// Device/Application/CheckFunctions/CheckBounds
// Short description:      Test function to increase machine safety by checking for unauthorized array indices accesses.
// 
// Functional description: This function is implicitly called prior to each array access and verifies if the access is within the valid array bounds.
//                         If the access is authorized, the function returns the index to the calling POU and the access is completed.
//                         If the access is unauthorized, an exception is triggered as default error reaction. This exception results in an application stop and the system is set to safe state. 
//   
// Handling particularities: Sporadically, the implemented default error reaction has TO be adjusted TO the application. 
//                           For example, stopping of the application can be invalid and can result in complicated recommissioning or even injury to people or damage to machines.
//                           Thus, adjust the default error reaction to your application.
//                           After inserting/removing this function in/from the project, no online change is possible.
//                           A complete download is required.
// 
// Further information:    The implicit calls of this check function are realized in all POUs but not in POUs of protected (*.compiled library) 
//                         and open (*.library) libraries or in POUs with the attribute {attribute 'no_check'}. Consequently, they do not increase the runtime.
//                         If the check is also to be performed in open libraries, enter the compiler definition 
//                         checks_in_libs in the field Compiler-Defines of the Build tab in the property dialog of the application node.
//                         An increased runtime depends on the number of programmed array accesses.
// 
//                         To reduce task runtimes, add the attribute 'no_check' to the POUs. 
//                         Checks performed by the check functions (CheckPointer, CheckBounds, CheckDiv, CheckRange) are not performed in these POUs. 
//                         Thus, these POUs have to be checked by the user regarding pointer programming, divisions and array accesses.  
//                         For more information, refer to the F1-help.
// 
//                         In the standard implementation, it is checked if the array access takes place within the valid array boundaries.
// 
//                         In case of invalid access (outside the valid array boundaries), an error is entered in the PLC logger and the application is stopped to avoid injury to persons and damage to machines.
//                         In this case, check the callstack (menu Debug/Callstack) and change the incorrect logic.
//
//                         If your application is not time-critical, use this function during commissioning as well as during the production phase of the machine.
//                         Only remove this function if you are sure that your user code is free from errors!
// 
// Do not change the declaration of this function! Add only local variables.  
// Do not change the attributes above the function header!
{attribute 'check_bounds'}
{attribute 'no_check'}
{attribute 'signature_flag' := '1073741824'}
FUNCTION CheckBounds : DINT
VAR_INPUT
  index, lower, upper: DINT;   // Index of the array, lower bound and upper bound
END_VAR
VAR
  ptNull: POINTER TO BYTE :=0; // Nullpointer for triggering an access violation
  strError: STRING;            // Diagnostic text for the PLC logger entry
END_VAR

    (*****************************************************************************************************)
    (* The implementation has to be adjusted to your application/machine.                                *)
    (* This is an exemplary implementation of the function.                                              *)
    (* Per default, an access violation is generated in case of an faulty acces to avoid machine damage. *)
    (* In this case, check the Call Stack (menu Debug/Callstack) and modify the faulty logic.            *)
    (*****************************************************************************************************)

IF  index < lower THEN 
  strError:= 'CheckBounds: Lower arrayindex ';
  strError:=CONCAT(STR1:=strError  , STR2:= DINT_TO_STRING(lower));
  strError:=CONCAT(STR1:=strError  , STR2:= ' underrunned by ');
  strError:=CONCAT(STR1:=strError  , STR2:= DINT_TO_STRING(index));
//  Default implementation for APPLICATION WILL BE STOPPED: 
//  Set an error into the plc logger
  LogAdd2(hLogger:= CmpLog.LOG_STD_LOGGER,udiCmpID:= 16#1000,udiClassID:= LogClass.LOG_ERROR,udiErrorID:= 1,udiInfoID:= 1,pszInfo:= strError);
//  Triggering an access violation --> Application will be stopped
  ptNull^ := 0;(* Triggering an access violation *)

// // Example for APPLICATION WILL NOT BE STOPPED:
// // Limit the faulty index to the lower index 
// //     --> no memory will be overwritten
// //     --> Keep PLC-task running
// // Set a warning into the plc logger
// // NOTE: There is still an implementation error in your application code!
// //  LogAdd2(hLogger:= CmpLog.LOG_STD_LOGGER,udiCmpID:= 16#1000,udiClassID:= LogClass.LOG_WARNING,udiErrorID:= 1,udiInfoID:= 1,pszInfo:= strError);
// // 
//  CheckBounds := lower; //access to the lower index only 
//  return;

ELSIF  index > upper THEN
  strError:= 'CheckBounds: Higher arrayindex ';
  strError:=CONCAT(STR1:=strError  , STR2:= DINT_TO_STRING(upper));
  strError:=CONCAT(STR1:=strError  , STR2:= ' overrunned by ');
  strError:=CONCAT(STR1:=strError  , STR2:= DINT_TO_STRING(index));

//  Default implementation for APPLICATION WILL BE STOPPED: 
//  Set an error into the plc logger
  LogAdd2(hLogger:= CmpLog.LOG_STD_LOGGER,udiCmpID:= 16#1000,udiClassID:= LogClass.LOG_ERROR,udiErrorID:= 1,udiInfoID:= 1,pszInfo:= strError);
//  Triggering an access violation --> Application will be stopped
  ptNull^ := 0;(* Triggering an access violation *)

// // Example for APPLICATION WILL NOT BE STOPPED:
// // Limit the faulty index to the upper index 
// //     --> no memory will be overwritten
// //     --> Keep PLC-task running
// // Set a warning into the plc logger
// // NOTE: There is still an implementation error in your application code!
//  LogAdd2(hLogger:= CmpLog.LOG_STD_LOGGER,udiCmpID:= 16#1000,udiClassID:= LogClass.LOG_WARNING,udiErrorID:= 1,udiInfoID:= 1,pszInfo:= strError);
// 
//  CheckBounds := upper; //access to the upper index only 
//  return;

ELSE // access to array is within lower and upper index --> ok  
  CheckBounds := index;
END_IF

END_FUNCTION

// Device/Application/CheckFunctions/CheckPointer
// Short description:      Test function to increase machine safety by detecting unauthorized accesses via POINTER and REFERENCE variables
//
// Functional description: This function is implicitly called prior to each pointer access and verifies if the access is invalid to 0.
//                         If the access is authorized, the function returns the pointer to the calling POU and the access is completed.
//                         If the access is unauthorized, an exception is triggered as default error reaction. This exception results in an application stop and the system is set to safe state. 
//                         It is recommended to adapt an appropriate error response to the machine application.
//   
// Handling particularities: Sporadically, the implemented default error reaction has to be adjusted to the application. 
//                           For example, stopping of the application can be invalid and can result in complicated recommissioning or even injury to people or damage to machines.
//                           Thus, adjust the default error reaction to your application.
//                           After inserting/removing this function in/from the project, no online change is possible.
//                           A complete download is required.
//                         
// Further information:    The implicit calls of this check function are realized in all POUs but not in POUs of protected (*.compiled library) 
//                         and open (*.library) libraries or in POUs with the attribute {attribute 'no_check'}. Consequently, they do not increase the runtime.
//                         If the check is also to be performed in open libraries, enter the compiler definition 
//                         checks_in_libs in the field Compiler-Defines of the Build tab in the property dialog of the application node.
//                         An increased runtime depends on the number of programmed pointer accesses or the use of REFERENCE variables.
//                         
//                         To reduce task runtimes, add the attribute 'no_check' to the POUs. 
//                         Checks performed by the check functions (CheckPointer, CheckBounds, CheckDiv, CheckRange) are not performed in these POUs. 
//                         Thus, these POUs have to be checked by the user regarding pointer programming, divisions and array accesses.  
//                         For more information, refer to the F1-help.
//                         
//                         In the standard implementation, it is checked if the pointer access takes place to Adress 16#0 (NULL-Pointer).
//                         In this case, check the callstack (menu Debug/Callstack) and change the incorrect logic.
//                         
//                         If your application is not time-critical, use this function during commissioning as well as during the production phase of the machine.
//                         Only remove this function if you are sure that your user code is free from errors!
//
// Do not change the declaration of this function! Add only local variables.  
// Do not change the attributes above the function header!
{attribute 'check_pointer'}
{attribute 'signature_flag' := '1073741824'}
{attribute 'no_check'}
FUNCTION CheckPointer : POINTER TO BYTE
VAR_INPUT 
  ptToTest : POINTER TO BYTE; // Pointer target address
  iSize : DINT;		            // Size of the type to which the pointer points. (z.B.: 20 für POINTER TO ARRAY [1..10] OF WORD) 
  iGran : DINT;		            // Granularity of the pointer access. This is the size of the largest unstructured data type in the type to which the pointer points. 
                                // (e.g.: 2 for POINTER TO ARRAY [0..9] OF INT).
  bWrite: BOOL;		            // Indicates read or write access. TRUE = write access.
END_VAR
VAR
  ptNull:   POINTER TO BYTE := 0; // Nullpointer for triggering an access violation
  strError: STRING(128);          // Diagnostic text for the PLC logger entry
  i: INT;						              // Index variable
END_VAR

IF ptToTest = 0 THEN //Just check NULL-Pointer

  IF bWrite THEN // write access
    strError:='CheckPointer: Invalid write-access to 16#0';
  ELSE
    strError:='CheckPointer: Invalid read-access to 16#0';
  END_IF
  strError:=CONCAT(STR1:=strError  , STR2:= ' - Size: ');
  strError:=CONCAT(STR1:=strError  , STR2:=TO_STRING(iSize));
  strError:=CONCAT(STR1:=strError  , STR2:=' - See callstack for reason!');
  
  LogAdd2(hLogger:= CmpLog.LOG_STD_LOGGER,udiCmpID:= 16#1000,udiClassID:= LogClass.LOG_ERROR,udiErrorID:= 1,udiInfoID:= 1,pszInfo:= strError);
  //  Triggering an access violation --> Application will be stopped
  //  Sporadically, this default error reaction has to be adjusted to the application. 
  //  For example, stopping of the application can be invalid and can result in complicated recommissioning or even injury to people or damage to machines.
  //  Thus, adjust the default error reaction to your application.
  ptNull^ := 0; //Triggering an access violation 
	
ELSE // pointer is not a NULL-Pointer
	CheckPointer := ptToTest; 
END_IF

END_FUNCTION

// Device/Application/CheckFunctions/CheckDivDInt
// Short description:        Test function to increase machine safety by detecting unauthorized division by zero of INT, UINT, DINT, UDINT, WORD and DWORD variables
// 
// Functional description:   This function will be called implicitly before the division takes places.
//                           The divisor will be checked for 0.
//                           In case of 0, an error is entered in the plc logger and the application is stopped due to an access violation to avoid machine damage.
//                           In this case, check the callstack (menu Debug/Callstack) and modify the faulty logic. 
// 
// Handling particularities: This function increases the cycle time of all tasks using divisions.
//                           The increase depends on the number of the divisions.
//                           After inserting/removing this function, no online-change will be possible! 
//                           A complete download will be necessary!
//                           The implementation has to be adjusted to your application/machine.
//                           In case of a division by zero, the PLC-Task will generate an access violation which leads to an application stop.
//                           Please verify whether this default behaviour can damage your machine or lead to a complex recommissioning. 
//                           In this case, adapt the error reaction to your application.
//                          
//                           If your application isn't too time-critical, you should leave this function whil comissioning the machine and production in your application.  
//                           If you remove this function, ensure that your code is faultless.
//                          
// Do not change the declaration of this function! Add only local variables.  
// Do not change the attributes above the function header!
{attribute 'check_div_int32'}
{attribute 'no_check'}
{attribute 'signature_flag' := '1073741824'}
FUNCTION CheckDivDInt : DINT
VAR_INPUT
  divisor: DINT; // Divisor of the division
END_VAR
VAR
  ptNull: POINTER TO BYTE := 0; // Nullpointer for triggering an access violation
  strError: STRING;             // Diagnostic text for the PLC logger entry
END_VAR

    (**************************************************************************************************)
    (* The implementation has to be adjusted to your application/machine.                             *)
    (* This is an exemplary implementation of the function.                                           *)
    (* Per default, an access violation is generated to avoid machine damage                          *)
    (* Check the Call Stack (menu Debug/Callstack) and modify the faulty logic!                       *)
    (**************************************************************************************************)

IF divisor = 0 THEN
  strError:= 'CheckDivDInt: Invalid division by 0 - check the callstack';
//  Default implementation for APPLICATION WILL BE STOPPED: 
//  Set an error into the plc logger
  LogAdd2(hLogger:= CmpLog.LOG_STD_LOGGER,udiCmpID:= 16#1000,udiClassID:= LogClass.LOG_ERROR,udiErrorID:= 1,udiInfoID:= 1,pszInfo:= strError);
//  Triggering an access violation --> Application will be stopped
  ptNull^ := 0;(* Triggering an access violation *)

// // Example for APPLICATION WILL NOT BE STOPPED:
// // Set the divisor to 1 
// //   --> no access violation (div by zero) will be triggered
// //   --> keep PLC-task running 
// // Set a warning into the plc logger
// // NOTE: There is still an implementation error in your application code!
// 
//  LogAdd2(hLogger:= CmpLog.LOG_STD_LOGGER,udiCmpID:= 16#1000,udiClassID:= LogClass.LOG_WARNING,udiErrorID:= 1,udiInfoID:= 1,pszInfo:= strError);
//  CheckDivDint := 1; //Division by 1 instead of zero 
//  return;	

ELSE // division is ok
  CheckDivDInt:=divisor;
END_IF;

END_FUNCTION

// Device/Application/CheckFunctions/CheckDivLInt
// Short description:        Test function to increase machine safety by detecting unauthorized division by zero of LINT, ULINT and LWORD variables
// 
// Functional description:   This function will be called implicitly before the division takes places.
//                           The divisor will be checked for 0.
//                           In case of 0, an error is entered in the plc logger and the application is stopped due to an access violation to avoid machine damage.
//                           In this case, check the callstack (menu Debug/Callstack) and modify the faulty logic. 
// 
// Handling particularities: This function increases the cycle time of all tasks using divisions.
//                           The increase depends on the number of the divisions.
//                           After inserting/removing this function, no online-change will be possible! 
//                           A complete download will be necessary!
//                           The implementation has to be adjusted to your application/machine.
//                           In case of a division by zero, the PLC-Task will generate an access violation which leads to an application stop.
//                           Please verify whether this default behaviour can damage your machine or lead to a complex recommissioning. 
//                           In this case, adapt the error reaction to your application.
//                          
//                           If your application isn't too time-critical, you should leave this function whil comissioning the machine and production in your application.  
//                           If you remove this function, ensure that your code is faultless.
//                          
// Do not change the declaration of this function! Add only local variables.  
// Do not change the attributes above the function header!
{attribute 'check_div_int64'}
{attribute 'no_check'}
{attribute 'signature_flag' := '1073741824'}
FUNCTION CheckDivLInt : LINT
VAR_INPUT
  divisor: LINT; // Divisor of the division
END_VAR
VAR
  ptNull: POINTER TO BYTE := 0; // Nullpointer for triggering an access violation
  strError: STRING;             // Diagnostic text for the PLC logger entry
END_VAR

    (**************************************************************************************************)
    (* The implementation has to be adjusted to your application/machine.                             *)
    (* This is an exemplary implementation of the function.                                           *)
    (* Per default, an access violation is generated to avoid machine damage                          *)
    (* Check the Call Stack (menu Debug/Callstack) and modify the faulty logic!                       *)
    (**************************************************************************************************)

IF divisor = 0 THEN
  strError:= 'CheckDivLInt: Invalid division by 0 - check the callstack';
//  Default implementation for APPLICATION WILL BE STOPPED: 
//  Set an error into the plc logger
  LogAdd2(hLogger:= CmpLog.LOG_STD_LOGGER,udiCmpID:= 16#1000,udiClassID:= LogClass.LOG_ERROR,udiErrorID:= 1,udiInfoID:= 1,pszInfo:= strError);
//  Triggering an access violation --> Application will be stopped
  ptNull^ := 0;(* Triggering an access violation *)

// // Example for APPLICATION WILL NOT BE STOPPED:
// // Set the divisor to 1 
// //   --> no access violation (div by zero) will be triggered
// //   --> keep PLC-task running 
// // Set a warning into the plc logger
// // NOTE: There is still an implementation error in your application code!
//  
//  LogAdd2(hLogger:= CmpLog.LOG_STD_LOGGER,udiCmpID:= 16#1000,udiClassID:= LogClass.LOG_WARNING,udiErrorID:= 1,udiInfoID:= 1,pszInfo:= strError);
//  CheckDivLInt := 1; //Division by 1 instead of zero 
//  return;	

ELSE // division is ok
  CheckDivLInt:=divisor;
END_IF;

END_FUNCTION

// Device/Application/CheckFunctions/CheckDivLReal
// Short description:        Test function to increase machine safety by detecting unauthorized division by zero of variables of type LREAL
// 
// Functional description:   This function will be called implicitly before the division takes places.
//                           The divisor will be checked for 0.0.
//                           In case of 0.0, an error is entered in the plc logger and the application is stopped due to an access violation to avoid machine damage.
//                           In this case, check the callstack (menu Debug/Callstack) and modify the faulty logic. 
// 
// Handling particularities: This function increases the cycle time of all tasks using divisions.
//                           The increase depends on the number of the divisions.
//                           After inserting/removing this function, no online-change will be possible! 
//                           A complete download will be necessary!
//                           The implementation has to be adjusted to your application/machine.
//                           In case of a division by zero, the PLC-Task will generate an access violation which leads to an application stop.
//                           Please verify whether this default behaviour can damage your machine or lead to a complex recommissioning. 
//                           In this case, adapt the error reaction to your application.
//                          
//                           If your application isn't too time-critical, you should leave this function whil comissioning the machine and production in your application.  
//                           If you remove this function, ensure that your code is faultless.
//                          
// Do not change the declaration of this function! Add only local variables.  
// Do not change the attributes above the function header!
{attribute 'check_div_real64'}
{attribute 'no_check'}
{attribute 'signature_flag' := '1073741824'}
FUNCTION CheckDivLReal : LREAL
VAR_INPUT
  divisor: LREAL; // Divisor of the division
END_VAR
VAR
  ptNull: POINTER TO BYTE := 0; // Nullpointer for triggering an access violation
  strError: STRING;             // Diagnostic text for the PLC logger entry
END_VAR

    (**************************************************************************************************)
    (* The implementation has to be adjusted to your application/machine.                             *)
    (* This is an exemplary implementation of the function.                                           *)
    (* Per default, an access violation is generated to avoid machine damage                          *)
    (* Check the Call Stack (menu Debug/Callstack) and modify the faulty logic!                       *)
    (**************************************************************************************************)

IF divisor = 0 THEN
  strError:= 'CheckDivLReal: Invalid division by 0 - check the callstack';
//  Default implementation for APPLICATION WILL BE STOPPED: 
//  Set an error into the plc logger
  LogAdd2(hLogger:= CmpLog.LOG_STD_LOGGER,udiCmpID:= 16#1000,udiClassID:= LogClass.LOG_ERROR,udiErrorID:= 1,udiInfoID:= 1,pszInfo:= strError);
//  Triggering an access violation --> Application will be stopped
  ptNull^ := 0;(* Triggering an access violation *)

// // Example for APPLICATION WILL NOT BE STOPPED:
// // Set the divisor to 1.0 
// //   --> no access violation (div by zero) will be triggered
// //   --> keep PLC-task running 
// // Set a warning into the plc logger
// // NOTE: There is still an implementation error in your application code!
//
//  LogAdd2(hLogger:= CmpLog.LOG_STD_LOGGER,udiCmpID:= 16#1000,udiClassID:= LogClass.LOG_WARNING,udiErrorID:= 1,udiInfoID:= 1,pszInfo:= strError);
//  CheckDivLReal := 1.0; //Division by 1 instead of zero 
//  return;	

ELSE // division is ok
  CheckDivLReal:=divisor;
END_IF;

END_FUNCTION

// Device/Application/CheckFunctions/CheckDivReal
// Short description:        Test function to increase machine safety by detecting unauthorized division by zero of variables of type REAL. 
// 
// Functional description:   This function will be called implicitly before the division takes places.
//                           The divisor will be checked for 0.0.
//                           In case of 0.0, an error is entered in the plc logger and the application is stopped due to an access violation to avoid machine damage.
//                           In this case, check the callstack (menu Debug/Callstack) and modify the faulty logic. 
// 
// Handling particularities: This function increases the cycle time of all tasks using divisions.
//                           The increase depends on the number of the divisions.
//                           After inserting/removing this function, no online-change will be possible! 
//                           A complete download will be necessary!
//                           The implementation has to be adjusted to your application/machine.
//                           In case of a division by zero, the PLC-Task will generate an access violation which leads to an application stop.
//                           Please verify whether this default behaviour can damage your machine or lead to a complex recommissioning. 
//                           In this case, adapt the error reaction to your application.
//                          
//                           If your application isn't too time-critical, you should leave this function whil comissioning the machine and production in your application.  
//                           If you remove this function, ensure that your code is faultless.
//                          
// Do not change the declaration of this function! Add only local variables.  
// Do not change the attributes above the function header!
{attribute 'check_div_real32'}
{attribute 'no_check'}
{attribute 'signature_flag' := '1073741824'}
FUNCTION CheckDivReal : REAL
VAR_INPUT
  divisor: REAL; // Divisor of the division
END_VAR
VAR
  ptNull: POINTER TO BYTE := 0; // Nullpointer for triggering an access violation
  strError: STRING;             // Diagnostic text for the PLC logger entry
END_VAR

    (**************************************************************************************************)
    (* The implementation has to be adjusted to your application/machine.                             *)
    (* This is an exemplary implementation of the function.                                           *)
    (* Per default, an access violation is generated to avoid machine damage                          *)
    (* Check the Call Stack (menu Debug/Callstack) and modify the faulty logic!                       *)
    (**************************************************************************************************)

IF divisor = 0 THEN
  strError:= 'CheckDivReal: Invalid division by 0 - check the callstack';
//  Default implementation for APPLICATION WILL BE STOPPED: 
//  Set an error into the plc logger
  LogAdd2(hLogger:= CmpLog.LOG_STD_LOGGER,udiCmpID:= 16#1000,udiClassID:= LogClass.LOG_ERROR,udiErrorID:= 1,udiInfoID:= 1,pszInfo:= strError);
//  Triggering an access violation --> Application will be stopped
  ptNull^ := 0;(* Triggering an access violation *)

// // Example for APPLICATION WILL NOT BE STOPPED:
// // Set the divisor to 1 
// //   --> no access violation (div by zero) will be triggered
// //   --> keep PLC-task running 
// // Set a warning into the plc logger
// // NOTE: There is still an implementation error in your application code!
// 
//  LogAdd2(hLogger:= CmpLog.LOG_STD_LOGGER,udiCmpID:= 16#1000,udiClassID:= LogClass.LOG_WARNING,udiErrorID:= 1,udiInfoID:= 1,pszInfo:= strError);
//  CheckDivReal := 1.0; //Division by 1 instead of zero 
//  return;	

ELSE // division is ok
  CheckDivReal:=divisor;
END_IF;

END_FUNCTION

// Device/Application/CheckFunctions/CheckLRangeSigned
// Short description:        Test function to increase machine safety by checking if value is within signed range (LINT) 
// 
// Functional description:  This function will be called implicitly before any access to range signed values.
//                           In case of invalid access, an error is entered in the diagnostic logbook and the application is stopped due to an access violation to avoid machine damage.
//                           In this case, check the callstack (menu Debug/Callstack) and modify the faulty logic. 
//                          
// Handling particularities: This function increases the cycle time of all tasks accessing range signed values. 
//                           The increase depends on the number of the read/write accesses.
// 
//                           After inserting/removing this function, no online-change will be possible! 
//                           A complete download will be necessary!
//                           The implementation has to be adjusted to your application/machine.
//                           In case of a division by zero, the PLC-Task will generate an access violation which leads to an application stop.
//                           Please verify whether this default behaviour can damage your machine or lead to a complex recommissioning. 
//                           In this case, adapt the error reaction to your application.
//
//                           If your application isn't too time-critical, you should leave this function whil comissioning the machine and production in your application.  
//                           If you remove this function, ensure that your code is faultless.
//                          
// Do not change the declaration of this function! Add only local variables.  
// Do not change the attributes above the function header!
{attribute 'no_check'}
{attribute 'check_lrange_signed'}
{attribute 'signature_flag' := '1073741824'}
FUNCTION CheckLRangeSigned : LINT
VAR_INPUT
  value: LINT;
  lower: LINT;
  upper: LINT;
END_VAR
VAR
  ptNull: POINTER TO BYTE := 0; // Nullpointer for triggering an access violation
  strError: STRING;             // Diagnostic text for the PLC logger entry
END_VAR

    (**************************************************************************************************)
    (* The implementation has to be adjusted to your application/machine.                             *)
    (* This is an exemplary implementation of the function.                                           *)
    (* Per default, an access violation is generated to avoid machine damage                          *)
    (* Check the Call Stack (menu Debug/Callstack) and modify the faulty logic!                       *)
    (**************************************************************************************************)

IF (value < lower) THEN
  strError:= 'CheckLRangeSigned: Lower value ';
  strError:=CONCAT(STR1:=strError  , STR2:= LINT_TO_STRING(lower));
  strError:=CONCAT(STR1:=strError  , STR2:= ' underrunned by ');
  strError:=CONCAT(STR1:=strError  , STR2:= LINT_TO_STRING(value));
//  Default implementation for APPLICATION WILL BE STOPPED: 
//  Set an error into the plc logger
  LogAdd2(hLogger:= CmpLog.LOG_STD_LOGGER,udiCmpID:= 16#1000,udiClassID:= LogClass.LOG_ERROR,udiErrorID:= 1,udiInfoID:= 1,pszInfo:= strError);
//  Triggering an access violation --> Application will be stopped
  ptNull^ := 0;(* Triggering an access violation *)

// // Example for APPLICATION WILL NOT BE STOPPED:
// // Limit the faulty value to the lower value 
// // Set a warning into the plc logger
// // NOTE: There is still an implementation error in your application code!
//
//	LogAdd2(hLogger:= CmpLog.LOG_STD_LOGGER,udiCmpID:= 16#1000,udiClassID:= LogClass.LOG_WARNING,udiErrorID:= 1,udiInfoID:= 1,pszInfo:= strError);
// 	CheckLRangeSigned := lower; //set value to lower value
//  return;
  
ELSIF(value > upper) THEN
  strError:= 'CheckLRangeSigned: Upper value ';
  strError:=CONCAT(STR1:=strError  , STR2:= LINT_TO_STRING(upper));
  strError:=CONCAT(STR1:=strError  , STR2:= ' overrunned by ');
  strError:=CONCAT(STR1:=strError  , STR2:= LINT_TO_STRING(value));

//  Default implementation for APPLICATION WILL BE STOPPED: 
//  Set an error into the plc logger
  LogAdd2(hLogger:= CmpLog.LOG_STD_LOGGER,udiCmpID:= 16#1000,udiClassID:= LogClass.LOG_ERROR,udiErrorID:= 1,udiInfoID:= 1,pszInfo:= strError);
//  Triggering an access violation --> Application will be stopped
  ptNull^ := 0;(* Triggering an access violation *)

// // Example for APPLICATION WILL NOT BE STOPPED:
// // Limit the faulty value to the upper value 
// // Set a warning into the plc logger
// // NOTE: There is still an implementation error in your application code!
// 
//  LogAdd2(hLogger:= CmpLog.LOG_STD_LOGGER,udiCmpID:= 16#1000,udiClassID:= LogClass.LOG_WARNING,udiErrorID:= 1,udiInfoID:= 1,pszInfo:= strError);
//  CheckLRangeSigned := upper; //set value to upper value
//  return;	

ELSE // value ist within valid range
  CheckLRangeSigned := value;
END_IF

END_FUNCTION

// Device/Application/CheckFunctions/CheckLRangeUnsigned
// Short description:        Test function to increase machine safety by checking if value is within unsigned range  (ULINT, LWORD) 
// 
// Functional description:   This function will be called implicitly before any access to range signed values.
//                           In case of invalid access, an error is entered in the diagnostic logbook and the application is stopped due to an access violation to avoid machine damage.
//                           In this case, check the callstack (menu Debug/Callstack) and modify the faulty logic. 
//                          
// Handling particularities: This function increases the cycle time of all tasks accessing range signed values. 
//                           The increase depends on the number of the read/write accesses.
// 
//                           After inserting/removing this function, no online-change will be possible! 
//                           A complete download will be necessary!
//                           The implementation has to be adjusted to your application/machine.
//                           In case of a division by zero, the PLC-Task will generate an access violation which leads to an application stop.
//                           Please verify whether this default behaviour can damage your machine or lead to a complex recommissioning. 
//                           In this case, adapt the error reaction to your application.
//                          
//                           If your application isn't too time-critical, you should leave this function whil comissioning the machine and production in your application.  
//                           If you remove this function, ensure that your code is faultless.
//                          
// Do not change the declaration of this function! Add only local variables.  
// Do not change the attributes above the function header!
{attribute 'no_check'}
{attribute 'check_lrange_unsigned'}
{attribute 'signature_flag' := '1073741824'}
FUNCTION CheckLRangeUnsigned : ULINT
VAR_INPUT
  value: ULINT;
  lower: ULINT;
  upper: ULINT;
END_VAR
VAR
  ptNull: POINTER TO BYTE := 0; // Nullpointer for triggering an access violation
  strError: STRING;             // Diagnostic text for the PLC logger entry
END_VAR

    (**************************************************************************************************)
    (* The implementation has to be adjusted to your application/machine.                             *)
    (* This is an exemplary implementation of the function.                                           *)
    (* Per default, an access violation is generated to avoid machine damage                          *)
    (* Check the Call Stack (menu Debug/Callstack) and modify the faulty logic!                       *)
    (**************************************************************************************************)

IF (value < lower) THEN
  strError:= 'CheckLRangeUnsigned: Lower value ';
  strError:=CONCAT(STR1:=strError  , STR2:= ULINT_TO_STRING(lower));
  strError:=CONCAT(STR1:=strError  , STR2:= ' underrunned by ');
  strError:=CONCAT(STR1:=strError  , STR2:= ULINT_TO_STRING(value));
//  Default implementation for APPLICATION WILL BE STOPPED: 
//  Set an error into the plc logger
  LogAdd2(hLogger:= CmpLog.LOG_STD_LOGGER,udiCmpID:= 16#1000,udiClassID:= LogClass.LOG_ERROR,udiErrorID:= 1,udiInfoID:= 1,pszInfo:= strError);
//  Triggering an access violation --> Application will be stopped
  ptNull^ := 0;(* Triggering an access violation *)

// // Example for APPLICATION WILL NOT BE STOPPED:
// // Limit the faulty value to the lower value 
// // Set a warning into the plc logger
// // NOTE: There is still an implementation error in your application code!
// 
//  CheckLRangeUnsigned := lower; //set value to lower value
//  return;

ELSIF(value > upper) THEN
  strError:= 'CheckLRangeUnsigned: Upper value ';
  strError:=CONCAT(STR1:=strError  , STR2:= ULINT_TO_STRING(upper));
  strError:=CONCAT(STR1:=strError  , STR2:= ' overrunned by ');
  strError:=CONCAT(STR1:=strError  , STR2:= ULINT_TO_STRING(value));

//  Default implementation for APPLICATION WILL BE STOPPED: 
//  Set an error into the plc logger
 LogAdd2(hLogger:= CmpLog.LOG_STD_LOGGER,udiCmpID:= 16#1000,udiClassID:= LogClass.LOG_ERROR,udiErrorID:= 1,udiInfoID:= 1,pszInfo:= strError);
//  Triggering an access violation --> Application will be stopped
 ptNull^ := 0;(* Triggering an access violation *)

// // Example for APPLICATION WILL NOT BE STOPPED:
// // Limit the faulty value to the upper value 
// // Set a warning into the plc logger
// // NOTE: There is still an implementation error in your application code!
// 
//  LogAdd2(hLogger:= CmpLog.LOG_STD_LOGGER,udiCmpID:= 16#1000,udiClassID:= LogClass.LOG_WARNING,udiErrorID:= 1,udiInfoID:= 1,pszInfo:= strError);
//  CheckLRangeUnsigned := upper; //set value to upper value
//  return;	

ELSE // value ist within valid range
  CheckLRangeUnsigned := value;
END_IF

END_FUNCTION

// Device/Application/CheckFunctions/CheckRangeSigned
// Short description:        Test function to increase machine safety by checking if value is within signed range (INT, DINT)  
// 
// Functional description:   This function will be called implicitly before any access to range signed values.
//                           In case of invalid access, an error is entered in the diagnostic logbook and the application is stopped due to an access violation to avoid machine damage.
//                           In this case, check the callstack (menu Debug/Callstack) and modify the faulty logic. 
//                          
// Handling particularities: This function increases the cycle time of all tasks accessing range signed values. 
//                           The increase depends on the number of the read/write accesses.
// 
//                           After inserting/removing this function, no online-change will be possible! 
//                           A complete download will be necessary!
//                           The implementation has to be adjusted to your application/machine.
//                           In case of a division by zero, the PLC-Task will generate an access violation which leads to an application stop.
//                           Please verify whether this default behaviour can damage your machine or lead to a complex recommissioning. 
//                           In this case, adapt the error reaction to your application.
//                          
//                           If your application isn't too time-critical, you should leave this function whil comissioning the machine and production in your application.  
//                           If you remove this function, ensure that your code is faultless.
//                          
// Do not change the declaration of this function! Add only local variables.  
// Do not change the attributes above the function header!
{attribute 'no_check'}
{attribute 'check_range_signed'}
{attribute 'signature_flag' := '1073741824'}
FUNCTION CheckRangeSigned : DINT
VAR_INPUT
  value: DINT;
  lower: DINT;
  upper: DINT;
END_VAR
VAR
  ptNull: POINTER TO BYTE := 0; // Nullpointer for triggering an access violation
  strError: STRING;             // Diagnostic text for the PLC logger entry
END_VAR

    (**************************************************************************************************)
    (* The implementation has to be adjusted to your application/machine.                             *)
    (* This is an exemplary implementation of the function.                                           *)
    (* Per default, an access violation is generated to avoid machine damage                          *)
    (* Check the Call Stack (menu Debug/Callstack) and modify the faulty logic!                       *)
    (**************************************************************************************************)

IF (value < lower) THEN
  strError:= 'CheckRangeSigned: Lower value ';
  strError:=CONCAT(STR1:=strError  , STR2:= DINT_TO_STRING(lower));
  strError:=CONCAT(STR1:=strError  , STR2:= ' underrunned by ');
  strError:=CONCAT(STR1:=strError  , STR2:= DINT_TO_STRING(value));
//  Default implementation for APPLICATION WILL BE STOPPED: 
//  Set an error into the plc logger
  LogAdd2(hLogger:= CmpLog.LOG_STD_LOGGER,udiCmpID:= 16#1000,udiClassID:= LogClass.LOG_ERROR,udiErrorID:= 1,udiInfoID:= 1,pszInfo:= strError);
//  Triggering an access violation --> Application will be stopped
  ptNull^ := 0;(* Triggering an access violation *)

// // Example for APPLICATION WILL NOT BE STOPPED:
// // Limit the faulty value to the lower value 
// // Set a warning into the plc logger
// // NOTE: There is still an implementation error in your application code!
//
//  LogAdd2(hLogger:= CmpLog.LOG_STD_LOGGER,udiCmpID:= 16#1000,udiClassID:= LogClass.LOG_WARNING,udiErrorID:= 1,udiInfoID:= 1,pszInfo:= strError);
//  CheckRangeSigned := lower; //set value to lower value
//  return;

ELSIF(value > upper) THEN
  strError:= 'CheckRangeSigned: Upper value ';
  strError:=CONCAT(STR1:=strError  , STR2:= DINT_TO_STRING(upper));
  strError:=CONCAT(STR1:=strError  , STR2:= ' overrunned by ');
  strError:=CONCAT(STR1:=strError  , STR2:= DINT_TO_STRING(value));

//  Default implementation for APPLICATION WILL BE STOPPED: 
//  Set an error into the plc logger
  LogAdd2(hLogger:= CmpLog.LOG_STD_LOGGER,udiCmpID:= 16#1000,udiClassID:= LogClass.LOG_ERROR,udiErrorID:= 1,udiInfoID:= 1,pszInfo:= strError);
//  Triggering an access violation --> Application will be stopped
  ptNull^ := 0;(* Triggering an access violation *)

// // Example for APPLICATION WILL NOT BE STOPPED:
// // Limit the faulty value to the upper value 
// // Set a warning into the plc logger
// // NOTE: There is still an implementation error in your application code!
// 
//  LogAdd2(hLogger:= CmpLog.LOG_STD_LOGGER,udiCmpID:= 16#1000,udiClassID:= LogClass.LOG_WARNING,udiErrorID:= 1,udiInfoID:= 1,pszInfo:= strError);
//  CheckRangeSigned := upper; //set value to upper value
//  return;	

ELSE // value ist within valid range
  CheckRangeSigned := value;
END_IF

END_FUNCTION

// Device/Application/CheckFunctions/CheckRangeUnsigned
// Short description:        Test function to increase machine safety by checking if value is within unsigned range (UINT, UDINT, WORD, DWORD)
// 
// Functional description:   This function will be called implicitly before any access to range unsigned values.
//                           In case of invalid access, an error is entered in the diagnostic logbook and the application is stopped due to an access violation to avoid machine damage.
//                           In this case, check the callstack (menu Debug/Callstack) and modify the faulty logic. 
//                          
// Handling particularities: This function increases the cycle time of all tasks accessing range signed values. 
//                           The increase depends on the number of the read/write accesses.
// 
//                           After inserting/removing this function, no online-change will be possible! 
//                           A complete download will be necessary!
//                           The implementation has to be adjusted to your application/machine.
//                           In case of a division by zero, the PLC-Task will generate an access violation which leads to an application stop.
//                           Please verify whether this default behaviour can damage your machine or lead to a complex recommissioning. 
//                           In this case, adapt the error reaction to your application.
//                          
//                           If your application isn't too time-critical, you should leave this function whil comissioning the machine and production in your application.  
//                           If you remove this function, ensure that your code is faultless.
//                          
// Do not change the declaration of this function! Add only local variables.  
// Do not change the attributes above the function header!
{attribute 'check_range_unsigned'}
{attribute 'signature_flag' := '1073741824'}
{attribute 'no_check'}
FUNCTION CheckRangeUnsigned : UDINT
VAR_INPUT
  value: UDINT;
  lower: UDINT;
  upper: UDINT;
END_VAR
VAR
  ptNull: POINTER TO BYTE := 0; // Nullpointer for triggering an access violation
  strError: STRING;             // Diagnostic text for the PLC logger entry
END_VAR

    (**************************************************************************************************)
    (* The implementation has to be adjusted to your application/machine.                             *)
    (* This is an exemplary implementation of the function.                                           *)
    (* Per default, an access violation is generated to avoid machine damage                          *)
    (* Check the Call Stack (menu Debug/Callstack) and modify the faulty logic!                       *)
    (**************************************************************************************************)

IF (value < lower) THEN
  strError:= 'CheckRangeUnsigned: Lower value ';
  strError:=CONCAT(STR1:=strError  , STR2:= UDINT_TO_STRING(lower));
  strError:=CONCAT(STR1:=strError  , STR2:= ' underrunned by ');
  strError:=CONCAT(STR1:=strError  , STR2:= UDINT_TO_STRING(value));
//  Default implementation for APPLICATION WILL BE STOPPED: 
//  Set an error into the plc logger
  LogAdd2(hLogger:= CmpLog.LOG_STD_LOGGER,udiCmpID:= 16#1000,udiClassID:= LogClass.LOG_ERROR,udiErrorID:= 1,udiInfoID:= 1,pszInfo:= strError);
//  Triggering an access violation --> Application will be stopped
  ptNull^ := 0;(* Triggering an access violation *)

// // Example for APPLICATION WILL NOT BE STOPPED:
// // Limit the faulty value to the lower value 
// // Set a warning into the plc logger
// // NOTE: There is still an implementation error in your application code!
//
//  LogAdd2(hLogger:= CmpLog.LOG_STD_LOGGER,udiCmpID:= 16#1000,udiClassID:= LogClass.LOG_WARNING,udiErrorID:= 1,udiInfoID:= 1,pszInfo:= strError);
//  CheckRangeUnsigned := lower; //set value to lower value
//  return;

ELSIF(value > upper) THEN
  strError:= 'CheckRangeUnsigned: Upper value ';
  strError:=CONCAT(STR1:=strError  , STR2:= UDINT_TO_STRING(upper));
  strError:=CONCAT(STR1:=strError  , STR2:= ' overrunned by ');
  strError:=CONCAT(STR1:=strError  , STR2:= UDINT_TO_STRING(value));

//  Default implementation for APPLICATION WILL BE STOPPED: 
//  Set an error into the plc logger
  LogAdd2(hLogger:= CmpLog.LOG_STD_LOGGER,udiCmpID:= 16#1000,udiClassID:= LogClass.LOG_ERROR,udiErrorID:= 1,udiInfoID:= 1,pszInfo:= strError);
//  Triggering an access violation --> Application will be stopped
 ptNull^ := 0;(* Triggering an access violation *)

// // Example for APPLICATION WILL NOT BE STOPPED:
// // Limit the faulty value to the upper value 
// // Set a warning into the plc logger
// // NOTE: There is still an implementation error in your application code!
// 
//  LogAdd2(hLogger:= CmpLog.LOG_STD_LOGGER,udiCmpID:= 16#1000,udiClassID:= LogClass.LOG_WARNING,udiErrorID:= 1,udiInfoID:= 1,pszInfo:= strError);
//  CheckRangeUnsigned := upper; //set value to upper value
//  return;

ELSE // value ist within valid range
  CheckRangeUnsigned := value;
END_IF

END_FUNCTION

// Device/Application/Json/FB_JsonDomParser
FUNCTION_BLOCK FB_JsonDomParser
VAR
 _parser : JsonParser2; 
END_VAR

METHOD CopyJson :UDINT
VAR_INPUT
  v    : POINTER TO JsonType;
  pDoc : POINTER to BYTE;
  nDoc : UDINT;
END_VAR
VAR
	Settings : JsonSerializeConfig;
END_VAR
CopyJson := TO_UDINT(JsonSerializer(v, pDoc,TO_DINT(nDoc),Settings));
END_METHOD

METHOD CopyString : UDINT
VAR_INPUT
  v    : POINTER TO JsonType;
  pStr : REFERENCE TO STRING;
  nStr : UDINT;
END_VAR
VAR_IN_OUT

END_VAR
VAR
	size: UDINT;
END_VAR
GetNodeAsString(v,ADR(pstr),nStr,retStrSize => size); 
CopyString := size;
END_METHOD

METHOD FindMember : POINTER TO JsonType; 
VAR_INPUT
  v      : POINTER TO JsonType;
END_VAR
VAR_IN_OUT CONSTANT
  member : STRING;
END_VAR
VAR
END_VAR
FindMember := GetJsonNodeByKey2(Member,v);
END_METHOD

METHOD GetArrayValueByIdx : POINTER TO JsonType
VAR_INPUT
  v   : POINTER TO JsonType;
  idx : UDINT;
END_VAR
GetArrayValueByIdx := GetNodeAtIndex(v,idx);
END_METHOD

METHOD GetBool : BOOL
VAR_INPUT
  v : POINTER TO JSONType;
END_VAR
VAR
	bValue :BOOL; 
	bSuccess: BOOL;
END_VAR
bSuccess := GetNodeAsBool(v,bJsonVal => bValue); 
GetBool := bValue and bSuccess;
END_METHOD

METHOD GetInt : DINT
VAR_INPUT
  v : POINTER TO JsonType;
END_VAR
VAR
	t_Dint: DINT;
	bSuccess: BOOL;
END_VAR
bSuccess := GetNodeAsInt(v,iJsonVal => t_Dint); 
IF bSuccess THEN 
	GetInt := t_Dint; 
END_IF
END_METHOD

METHOD GetString : STRING(255)
VAR_INPUT
  v : POINTER TO JsonType;
END_VAR
VAR
	bytes : ARRAY[0..256] OF BYTE; 
	pString : POINTER TO STRING(255); 
END_VAR
pString := ADR(bytes); 
GetNodeAsString(v,pString,256); 
GetString := pString^;
END_METHOD

METHOD ParseDocument : POINTER TO JsonType
VAR_INPUT
	udSize : UDINT;
END_VAR
VAR_IN_OUT CONSTANT
  sJson : STRING;
END_VAR
ParseDocument := 0; 
IF(_parser.Parse(ADR(sJson),udSize)) THEN 
	ParseDocument := _parser.GetRootDoc(); 
END_IF
END_METHOD

END_FUNCTION_BLOCK

// Device/Application/Json/FB_JsonSaxWriter
{attribute 'hide_all_locals'}
FUNCTION_BLOCK FB_JsonSaxWriter
VAR_INPUT
END_VAR
VAR_OUTPUT
	initStatus: POINTER TO JsonType;
END_VAR
VAR
	_arrObjects : ARRAY[0..JSONParameters.MAX_DOC_DEPTH] OF POINTER TO JsonObjectManager; 
	_arrArrays  : ARRAY[0..JSONParameters.MAX_DOC_DEPTH] OF POINTER TO DynamicList; 
	_objIdx : INT; 
	_arrIdx : INT; 
	_curArrIdx : ARRAY[0.. JSONParameters.MAX_DOC_DEPTH] OF UDINT;  
	_bArr : BOOL; 
	_Key  : POINTER TO BYTE; 
	_root : JsonType;
	_backingArCreatedVals : DynamicJsonTypeContainer(udSize := 1); 
	_lCreatedValues : DynamicList :=(DataContainer := _backingArCreatedVals); 
	_backingArCreatedObj : DynamicJsonObjectContainer(udSize := 1); 
	_lCreatedObj : DynamicList := (DataContainer := _backingArCreatedObj); 
	_backingArrayCreatedKeys : DynamicStringContainer(udSize := 1); 
	_lCreatedKeys: DynamicList := (DataContainer  := _backingArrayCreatedKeys);
	backingArrayArrays : DynamicJsonContainerContainer(udSize := 1);
	lCreatedLists : DynamicList := (DataContainer := backingArrayArrays);  
	_strRoot : STRING := 'root';
	_bInit : BOOL; 
	_AddKey: BOOL;
	_bRootAdded : BOOL; 
END_VAR

METHOD AddBool : BOOL
VAR_INPUT
  value : BOOL;
END_VAR
VAR
	pJsonType: POINTER TO JSONType;
	pBool: POINTER TO BOOL;
END_VAR
IF NOT _bInit AND NOT _barr AND NOT _AddKey THEN
	AddBool := FALSE; 
	RETURN; 
END_IF
pJsonType := CreateJsonType(); 
pJsonType^.DataType := JsonDataType.JSON_DATA_BOOL; 
pBool := __NEW(BOOL); 
pBool^ := value;
pJsonType^.pValue := pBool;  
IF NOT _bArr THEN 
	_arrObjects[_ObjIdx]^.Put(_key,pJsonType); 
  	_AddKey := FALSE; 
ELSE 
	_arrArrays[_arrIdx]^.PushBack(ADR(pJsonType)); 
END_IF
END_METHOD

METHOD AddDint : BOOL
VAR_INPUT
  value : DINT;
END_VAR

VAR
	pJson : POINTER TO JsonType;
	pDint: POINTER TO DINT;
END_VAR
IF NOT _bInit AND NOT _barr AND NOT _AddKey THEN 
	RETURN; 
END_IF
pJson := CreateJsonType(); 
pJson^.DataType := JSONDATATYPE.JSON_DATA_INT; 
pDint := __NEW(DINT); 
pDint^ := value;
pJson^.pValue := pDint; 
IF NOT _bArr THEN 
	_arrObjects[_objIdx]^.Put(_key,pJson); 
	_AddKey := FALSE; 
ELSE 
	_arrArrays[_arrIdx]^.PushBack(ADR(pJson)); 
END_IF
END_METHOD

METHOD AddKey : BOOL
VAR_IN_OUT CONSTANT
	key: STRING;
END_VAR

VAR

	_i: DINT;
END_VAR
_i := 0; 
WHILE Key[_i] <> 0 DO
	_i := _i + 1; 
END_WHILE
_i := _i + 1; 
_key := __NEW(BYTE,_i); 
_i := 0; 
WHILE Key[_i] <> 0 DO
	_key[_i] := key[_i]; 
	_i := _i + 1; 
END_WHILE
_key[_i] := 0; 
_lCreatedKeys.PushBack(ADR(_key)); 
_AddKey := TRUE; 
AddKey := TRUE;
END_METHOD

METHOD AddNull 
VAR_INPUT
END_VAR

VAR
	pJson: Pointer TO JsonTYpe;
END_VAR
IF NOT _bInit AND NOT _barr AND NOT _AddKey THEN 
	RETURN; 
END_IF
pJson := CreateJsonType(); 
pJson^.DataType := JSONDATATYPE.JSON_DATA_NULL; 
pJson^.pValue := 0; 
IF NOT _bArr THEN 
	_arrObjects[_objIdx]^.Put(_key,pJson); 
	_AddKey := FALSE; 
ELSE 
	_arrArrays[_arrIdx]^.PushBack(ADR(pJson)); 
END_IF
_AddKey := FALSE;
END_METHOD

METHOD AddString : BOOL
VAR_IN_OUT CONSTANT
	value: STRING;
END_VAR
VAR
	pJson : POINTER TO JsonType; 
	_i: INT;
	pString: POINTER TO BYTE;
END_VAR
IF NOT _bInit AND NOT _barr AND NOT _AddKey THEN 
	RETURN; 
END_IF
pJson := CreateJsonType(); 
pJson^.DataType := JSONDATATYPE.JSON_DATA_STRING; 
_i := 0;
WHILE value[_i] <> 0 DO
	_i := _i + 1; 
END_WHILE
pString := __NEW(BYTE,_i); 
_i := 0; 
WHILE value[_i] <> 0 DO 
	pString[_i] := value[_i]; 
	_i := _i + 1; 
END_WHILE
pString[_i] := 0; 
pJson^.pValue := pString; 
IF NOT _bArr THEN 
	_arrObjects[_objIdx]^.Put(_key,pJson); 
	_AddKey := FALSE; 
ELSE 
	_arrArrays[_arrIdx]^.PushBack(ADR(pJson)); 
END_IF
END_METHOD

METHOD AddUdint
VAR_INPUT
  value : UDINT;
END_VAR
VAR
	
	pJson: Pointer TO JsonType;
	pDint: POINTER TO UDINT;
END_VAR
IF NOT _bInit AND NOT _barr AND NOT _AddKey THEN 
	RETURN; 
END_IF
pJson := CreateJsonType(); 
pJson^.DataType := JSONDATATYPE.JSON_DATA_INT; 
pDint := __NEW(UDINT); 
pDint^ := value;
pJson^.pValue := pDint; 
IF NOT _bArr THEN 
	_arrObjects[_objIdx]^.Put(_key,pJson); 
	_AddKey := FALSE; 
ELSE 
	_arrArrays[_arrIdx]^.PushBack(ADR(pJson)); 
END_IF
END_METHOD

METHOD CopyDocument : UDINT
VAR_IN_OUT CONSTANT
  pDoc       : STRING;
END_VAR
VAR_INPUT
  nDoc       : UDINT;
  bPretty : BOOL := FALSE; 
END_VAR
VAR_OUTPUT
  hrErrorCode:PVOID;
END_VAR
VAR
	_bytePtr : POINTER TO BYTE; 
	_i: UDINT;
	_Settings : JsonSerializeConfig;
END_VAR
IF NOT _bInit THEN 
	Init(); 
END_IF
_bytePtr := ADR(pDoc); 
_settings.PrettyPrint := bPretty;
_settings.IndentSize := 4; 
CopyDocument := TO_UDINT(JsonSerializer(GetRoot(),ADR(pDoc),TO_DINT(nDoc),_settings));
END_METHOD

METHOD EndArray 
VAR_INPUT
END_VAR
IF NOT _bInit THEN
	Init(); 
END_IF
_arrIdx := _arrIdx - 1; 
IF _arrIdx < 0 THEN
	_bArr := FALSE; 
	_AddKey := FALSE; 
END_IF
END_METHOD

METHOD EndObject 
VAR_INPUT
END_VAR

VAR

END_VAR
IF NOT _bInit THEN
	Init(); 
END_IF
_AddKey := FALSE; 
_ObjIdx := _ObjIdx - 1;
END_METHOD

//FB_Exit must be implemented explicitly. If there is an implementation, then the
//method is called before the controller removes the code of the function block instance
//(implicit call). The return value is not evaluated.
METHOD FB_Exit: BOOL
VAR_INPUT
    bInCopyCode: BOOL;  // TRUE: the exit method is called in order to leave the instance which will be copied afterwards (online change).  
END_VAR
Clean();
END_METHOD

METHOD PRIVATE Init : BOOL
VAR_INPUT
END_VAR
_root.DataType := JSONDATATYPE.JSON_DATA_OBJECT; 
_root.pValue := CreateObj(); 
_arrObjects[0] := _root.pValue;  
_bInit := TRUE; 
_arrIdx := -1; 
_objIdx := 0;
_bRootAdded := FALSE;
END_METHOD

METHOD ResetDocument 
VAR_INPUT
END_VAR
Clean(); 
_bInit :=FALSE; 
_AddKey:=FALSE;
_bRootAdded :=FALSE; 
_arrIdx := -1; 
_objIdx := 0;
END_METHOD

METHOD StartArray  
VAR_INPUT
END_VAR
VAR
	pJson : POINTER TO JSONTYPE; 
	pArr: POINTER TO DynamicList;
END_VAR
IF NOT _bInit THEN
	Init(); 
END_IF
IF NOT _bRootAdded THEN 
	AddKey('root'); 
	_bRootAdded := TRUE; 
END_IF
IF NOT _barr AND NOT _AddKey THEN 
	RETURN; 
END_IF
_arrIdx := _arrIdx + 1; 
pJson := CreateJsonType(); 
pJson^.DataType := JSONDATATYPE.JSON_DATA_ARRAY; 
pArr := CreateArray();
pJson^.pValue := pArr; 
IF NOT _bArr THEN 
	_arrObjects[_objIdx]^.Put(_key,pJson); 
	_AddKey := FALSE; 
ELSE 
	_arrArrays[_arrIdx-1]^.PushBack(ADR(pJson)); 
END_IF
_arrArrays[_arrIdx] := pArr; 
_bArr := TRUE;
END_METHOD

METHOD StartObject 
VAR_INPUT
END_VAR

VAR

	pJson: POINTER TO JsonType;
	pObj: POINTER TO JsonObjectManager;
	pRoot: POINTER TO BYTE;
	strRoot : STRING := 'root'; 
END_VAR
IF NOT _bInit THEN
	Init(); 
END_IF
IF NOT _bRootAdded THEN 
	IF NOT _addKey THEN 
		AddKey('root'); 
		_bRootAdded := TRUE; 
	ELSE
		pJson := CreateJsonType(); 
		pJson^.DataType := JSONDATATYPE.JSON_DATA_OBJECT; 
		pObj:= CreateObj(); 
		pJson^.pValue := pObj; 
		pRoot := __NEW(BYTE,5); 
		pRoot[0] := strRoot[0];
		pRoot[1] := strRoot[1];
		pRoot[2] := strRoot[2];
		pRoot[3] :=strRoot[3];
		pRoot[4] :=0; 
		_lCreatedKeys.PushBack(ADR(pRoot)); 
		_arrObjects[_objIdx]^.Put(pRoot,pJson);
		_objIdx := _objIdx + 1; 
		_arrObjects[_objIdx] := pJson^.pValue; 
		_bRootAdded := TRUE; 
	END_IF
END_IF
IF NOT _barr AND NOT _AddKey THEN 
	RETURN; 
END_IF 
pJson := CreateJsonType(); 
pJson^.DataType := JSONDATATYPE.JSON_DATA_Object; 
pObj := CreateObj();
pJson^.pValue := pObj; 
IF NOT _bArr THEN 
	_arrObjects[_objIdx]^.Put(_key,pJson); 
	_AddKey := FALSE; 
ELSE 
	_arrArrays[_arrIdx]^.PushBack(ADR(pJson)); 
END_IF
_objIdx := _objIdx + 1; 
_arrObjects[_objIdx] := pObj;
END_METHOD

END_FUNCTION_BLOCK

// Device/Application/ResizableMem (Not Fully Tested)/DynamicQueue
{attribute 'no_check'}
{attribute 'enable_dynamic_creation'}
FUNCTION_BLOCK DynamicQueue IMPLEMENTS iQueue
VAR_INPUT
	DataContainer : iDynamicDataContainer; 
END_VAR
VAR_OUTPUT
END_VAR
VAR
	_size : UDINT; 
	_front: UDINT; 
	_backingSize : UDINT := 0; 
END_VAR

END_FUNCTION_BLOCK

// Device/Application/ResizableMem (Not Fully Tested)/JsonListManager
{attribute 'enable_dynamic_creation'}
FUNCTION_BLOCK JsonListManager 
VAR_INPUT
END_VAR
VAR
	_BackingValues : POINTER TO DynamicJsonTypeContainer; 
	_List          : POINTER TO DynamicList; 
END_VAR

METHOD Create : BOOL
VAR_INPUT
END_VAR
IF _BackingValues <> 0 THEN 
	RETURN; 
END_IF
_BackingValues := __NEW(DynamicJsonTypeCOntainer(udSize := 10, iDeleter := JsonHelpers.instDeleteJsonType)); 
_List := __NEW(DynamicList); 
_List^(DataContainer := _BackingValues);
END_METHOD

METHOD Destroy : BOOL
VAR_INPUT
END_VAR
IF _backingValues <> 0 THEN 
	__DELETE(_backingValues); 
END_IF
IF _List <> 0 THEN 
	__DELETE(_LIST); 
END_IF
END_METHOD

METHOD GetAt : POINTER TO JsonType
VAR_INPUT
	index : UDINT; 
END_VAR
VAR
	pJsonType : POINTER TO JsonType; 
END_VAR
pJsonType := 0; 
_List^.Get(index,ADR(pJsonType)); 
GetAt := pJsonType;
END_METHOD

METHOD Push : BOOL
VAR_INPUT
	pJson : POINTER TO JsonType; 
END_VAR
_List^.PushBack(ADR(pJson));
END_METHOD

END_FUNCTION_BLOCK

// Device/Application/Util/ADT_CompareString
FUNCTION_BLOCK ADT_CompareString Implements iCompare
VAR_INPUT
END_VAR
VAR_OUTPUT
END_VAR
VAR
END_VAR

(* Pointers to the data being comapred are passed, 
   Compare >0 Data1 > Data2 
   Compare <0 Data1 < Data2 
   Compare = 0 Data 1 = Data2 *)
METHOD Compare : INT
VAR_INPUT
	pData1	: PVoid;
	pData2	: PVoid;
END_VAR
VAR
	pString1 : POINTER TO POINTER TO STRING;  
	ppString2 : POINTER TO POINTER TO STRING;
END_VAR
pString1 := pData1; 
ppString2 := pData2;

IF pString1^^ = ppString2^^ THEN 
	Compare := 0; 
	RETURN;
END_IF
Compare := 1;
END_METHOD

END_FUNCTION_BLOCK

// Device/Application/Util/StringHash
{attribute 'no_check'}
FUNCTION_BLOCK StringHash IMPLEMENTS iHash
VAR_INPUT
END_VAR
VAR_OUTPUT
END_VAR
VAR
END_VAR

{attribute 'no_check'}
METHOD Hash : LINT
VAR_INPUT
	pData	: pVoid;
END_VAR
VAR
	ppString : POINTER TO POINTER TO STRING; 
	pString : POINTER TO STRING; 
	_i: INT;
	_multiple: LINT;
	_hash : LINT; 
END_VAR
_multiple := 1; 
_hash := 0; 
ppString := pData; 
pString := ppString^; 
FOR _i :=0 TO LEN(pString^) - 1 DO 
	_hash := _hash + pString^[_i] * _multiple; 
	_multiple := _multiple*97;
	IF _multiple > 760231058654565216 THEN 
		_multiple := 1; 
	END_IF  
END_FOR
Hash := _hash;
END_METHOD

END_FUNCTION_BLOCK
